IF rtInit.Q					//初始化确认窗口显示
	AND xEStop
	AND xSafety
	AND xManualMode
	AND NOT xAlarm
	AND NOT xIniting
THEN
	wWindow[nWindowNumberIndex]:=nInitConfirmWindow;
END_IF

IF rtInit.Q					//初始化有报警
	AND xAlarm
THEN
	wWindow[nWindowNumberIndex]:=nInitAlarmWindow;
END_IF

IF xIniting					//初始化中有报警
	AND xAlarm
THEN
	wWindow[nWindowNumberIndex]:=nInitingAlarmWindow;
END_IF

IF xIniting THEN			//初始化中窗口显示
	wWindow[nWindowNumberIndex]:=nInitingWindow;
END_IF

IF ftIniting.Q THEN		
	IF xInitDone THEN		//初始化完成窗口显示
		wWindow[nWindowNumberIndex]:=nInitDoneWindow;
	ELSE					//初始化失败窗口显示
		wWindow[nWindowNumberIndex]:=nInitFailWindow;
	END_IF
END_IF

IF xWindowColseHMI
THEN
	wWindow[nWindowNumberIndex]:=0;
	wWindow[nWindowControlIndex]:=0;
END_IF
END_ACTION

END_FUNCTION_BLOCK

// Device/Application/FB/14_MachineFB/FB_Machine_1
FUNCTION_BLOCK FB_Machine_1
VAR_INPUT
	CT_input           :BOOL;   //计时信号
	CT_number          :REAL:=1;//出料数量设定
	Sta_xtart_b        :BOOL;   //启动按钮
	Sta_xstop_b        :BOOL;   //停止按钮
	Sta_xreset_b       :BOOL;   //复位按钮
	Sta_safety         :BOOL;   //安全条件、
END_VAR
VAR_OUTPUT
	CT_TIME            :REAL;   //节拍时间
	Sta_xrunning       :BOOL;   //运行状态
	Sta_xstop          :BOOL;   //停止状态
	Sta_xiniting       :BOOL;   //初始化中
	Sta_xPaused        :BOOL;   //暂停中
	Sta_xEmptying      :BOOL;   //清料中（排空）
END_VAR
VAR_IN_OUT
END_VAR
VAR
	CT_Rtinput            : R_TRIG;         //计时信号上升沿
	CT_TEMP               : UDINT;
	CT_Start              : UDINT;
	CT_Stop               : UDINT;
END_VAR

ACTION ACT_CT:

//  CT计算
CT_Rtinput(CLK:= CT_input , Q=> );
IF Sta_xrunning AND CT_Rtinput.Q THEN
	 GetSystemTime(udiTimeMs=> CT_Stop, uliTimeUs=> , uliTimeNs=> );
	 IF CT_Start<>0 THEN
	 CT_TEMP := CT_Stop-CT_Start;
	 END_IF
	 CT_Start:=CT_Stop;
END_IF
IF NOT Sta_xrunning THEN
	CT_Stop :=0;
  CT_Start:=0;
	CT_TEMP :=0;
END_IF
CT_TIME:= (UDINT_TO_REAL(CT_TEMP)/1000.0)/CT_number;
END_ACTION

ACTION ACT_status:
IF Sta_safety THEN
   IF Sta_xtart_b THEN
	  Sta_xrunning:=TRUE;
   END_IF
END_IF
END_ACTION

END_FUNCTION_BLOCK

// Device/Application/FC_check/CheckBounds
// 隐含生成代码：不要编辑
FUNCTION CheckBounds : DINT
VAR_INPUT
	index, lower, upper: DINT;
END_VAR

// 隐含生成代码：这里只是对代码实现的建议
IF  index < lower THEN
	CheckBounds := lower;
ELSIF  index > upper THEN
	CheckBounds := upper;
ELSE  
	CheckBounds := index;
END_IF

(*还可以设置断点，日志消息或停止异常情况。
Add CmpApp.library, SysExcept.library and SysTypes2_Itf as newest.
Declaration:
VAR
    _pApp : POINTER TO CmpApp.APPLICATION;
    _result   : SysTypes.RTS_IEC_RESULT;
END_VAR

Implementation:
_pApp := AppGetCurrent(pResult:=_result);
IF  index < lower THEN
        CheckBounds := lower;
        IF _pApp <> 0 THEN
                AppGenerateException(pApp:=_pApp, ulException:=RtsExceptions.RTSEXCPT_ARRAYBOUNDS);
        END_IF
ELSIF  index > upper THEN
        CheckBounds := upper;
        IF _pApp <> 0 THEN
                AppGenerateException(pApp:=_pApp,   ulException:=RtsExceptions.RTSEXCPT_ARRAYBOUNDS);
        END_IF
ELSE  
        CheckBounds := index;
END_IF
*)

END_FUNCTION

// Device/Application/FC_check/CheckDivDInt
// 隐含生成代码：不要编辑
FUNCTION CheckDivDInt : DINT
VAR_INPUT
	divisor:DINT;
END_VAR

// 隐含生成代码：这里只是对代码实现的建议
IF divisor = 0 THEN
	CheckDivDInt:=1;
ELSE
	CheckDivDInt:=divisor;
END_IF;

END_FUNCTION

// Device/Application/FC_check/CheckDivLInt
// 隐含生成代码：不要编辑
FUNCTION CheckDivLInt : LINT
VAR_INPUT
	divisor:LINT;
END_VAR

// 隐含生成代码：这里只是对代码实现的建议
IF divisor = 0 THEN
	CheckDivLInt:=1;
ELSE
	CheckDivLInt:=divisor;
END_IF;

END_FUNCTION

// Device/Application/FC_check/CheckDivReal
// 隐含生成代码：不要编辑
FUNCTION CheckDivReal : REAL
VAR_INPUT
	divisor:REAL;
END_VAR

// 隐含生成代码：这里只是对代码实现的建议
IF divisor = 0 THEN
	CheckDivReal:=1;
ELSE
	CheckDivReal:=divisor;
END_IF;

END_FUNCTION

// Device/Application/FC_check/CheckDivLReal
// 隐含生成代码：不要编辑
FUNCTION CheckDivLReal : LREAL
VAR_INPUT
	divisor:LREAL;
END_VAR

// 隐含生成代码：这里只是对代码实现的建议
IF divisor = 0 THEN
	CheckDivLReal:=1;
ELSE
	CheckDivLReal:=divisor;
END_IF;

END_FUNCTION

// Device/Application/FC_check/CheckPointer
// 隐含生成代码：不要编辑
FUNCTION CheckPointer : POINTER TO BYTE
VAR_INPUT 
	ptToTest : POINTER TO BYTE; // 指针的目标地址
	iSize : DINT;		        // 指针指向的类型大小。（例如：POINTER TO ARRAY [0..9] OF INT为20）
	iGran : DINT;		        // 指针访问的粒度，即指针指向的类型中最大的非结构数据类型的大小。（例如：POINTER TO ARRAY [0..9] OF INT为2）
	bWrite: BOOL;		        // 指示读或写权限。TRUE=写权限。
END_VAR

// 没有标准的实现方式。在此处输入代码
CheckPointer := ptToTest;

END_FUNCTION

// Device/Application/FC_check/CheckRangeSigned
// 隐含生成代码：不要编辑
FUNCTION CheckRangeSigned : DINT
VAR_INPUT
	value, lower, upper: DINT;
END_VAR

// 隐含生成代码：这里只是对代码实现的建议
IF (value < lower) THEN
	CheckRangeSigned := lower;
ELSIF(value > upper) THEN
	CheckRangeSigned := upper;
ELSE
	CheckRangeSigned := value;
END_IF

END_FUNCTION

// Device/Application/FC_check/CheckRangeUnsigned
// 隐含生成代码：不要编辑
FUNCTION CheckRangeUnsigned : UDINT
VAR_INPUT
	value, lower, upper: UDINT;
END_VAR

// 隐含生成代码：这里只是对代码实现的建议
IF (value < lower) THEN
	CheckRangeUnsigned := lower;
ELSIF(value > upper) THEN
	CheckRangeUnsigned := upper;
ELSE
	CheckRangeUnsigned := value;
END_IF

END_FUNCTION

// Device/Application/FC_check/CheckLRangeSigned
// 隐含生成代码：不要编辑
FUNCTION CheckLRangeSigned : LINT
VAR_INPUT
	value, lower, upper: LINT;
END_VAR

// 隐含生成代码：这里只是对代码实现的建议
IF (value < lower) THEN
	CheckLRangeSigned := lower;
ELSIF(value > upper) THEN
	CheckLRangeSigned := upper;
ELSE
	CheckLRangeSigned := value;
END_IF

END_FUNCTION

// Device/Application/FC_check/CheckLRangeUnsigned
// 隐含生成代码：不要编辑
FUNCTION CheckLRangeUnsigned : ULINT
VAR_INPUT
	value, lower, upper: ULINT;
END_VAR

// 隐含生成代码：这里只是对代码实现的建议
IF (value < lower) THEN
	CheckLRangeUnsigned := lower;
ELSIF(value > upper) THEN
	CheckLRangeUnsigned := upper;
ELSE
	CheckLRangeUnsigned := value;
END_IF

END_FUNCTION
